{attribute 'qualified_only'}
VAR_GLOBAL
	Befehle: BYTE;
 	Ver: ARRAY[0..255] OF BYTE;
END_VAR

(* stored: Version 1.1.0.1, ProductVersion 3.1.4024.5
   GVL VersionsInfo: Id {6d3a9978-b91d-41da-a104-582bc67bc2a4} *)
